FUNCTION_BLOCK FB_4PVICI_EPS EXTENDS FB_4PortViciValve
VAR_INPUT
END_VAR
VAR_OUTPUT
	bAllPortsLocked : BOOL;
	bExternalLock : BOOL;
END_VAR
VAR_IN_OUT
	aPortEPS : ARRAY [1 .. 4] OF DUT_VICI_PORT_EPS; // EPS for each port.
END_VAR
VAR
	{attribute 'pytmc' := '
	pv: PORT
	io: o
	'}
	iNewPortPos : INT;
	
	{attribute 'pytmc' := 'pv: OVRD_MODE'}
    bEPS_Override : BOOL := FALSE;
    {attribute 'pytmc' := 'pv: OVRD_COUNTDOWN'}
    tEPS_TimerCountDown : STRING := TIME_TO_STRING(T#0s);
    fbTimer : TON;
	tEPS_OVRD_RESET_TIME : TIME := T#1m;

	
END_VAR

iReqPos := LIMIT(1,iReqPos, 4); // KEEP EPS array index within bounds

M_RESET_OVERRIDE_TIMER();

iNewPortPos := M_EPS_LOGIC(aPortEPS := aPortEPS, 
							iReqPort := iReqPos,
							iPrevPort := iNewPortPos,
							bOverride := FALSE,
							bExternalLockSignal => bExternalLock,
							bAllPortsLocked => bAllPortsLocked);

fbNporValve(iAddress := iAdress, 
			iNumOfPorts := iNumPorts, 
			iReqPos := iNewPortPos);
			


(*
Qs
- Should there be a valve to stop the flow if none of the EPS conditions are met?
- Should the VICI valve always go to a EPS condition that is true?


PORT ENUM
- LOCKED 	(EPS not OK)
- UNLOCKED 	(EPS OK but not active)
- ACTIVE	(EPS OK and ACTIVE)
*)

METHOD M_EPS_LOGIC : INT
VAR_INPUT
	iReqPort : INT;
	iPrevPort : INT;
	bOverride : BOOL;
END_VAR
VAR_IN_OUT
	aPortEPS : ARRAY [1 .. 4] OF DUT_VICI_PORT_EPS;
END_VAR
VAR_OUTPUT
	bAllPortsLocked : BOOL;
	bExternalLockSignal : BOOL; // Signal to external device that port is locked.
END_VAR
VAR
	fbEPS : FB_EPS;
	iIndex : INT := 1;
	iEPS_NOT_OK_COUNT : INT;
	iNewPortPos : INT;
END_VAR
// Evaluate all EPS 
FOR iIndex := 1 TO iNumPorts BY 1 DO
	
	fbEPS(eps := aPortEPS[iIndex].stEPS);
	
	IF aPortEPS[iIndex].stEPS.bEPS_OK THEN
		aPortEPS[iIndex].ePortStatus := ENUM_PORT_STATUS.UNLOCKED;
	ELSE
		aPortEPS[iIndex].ePortStatus := ENUM_PORT_STATUS.LOCKED;
		iEPS_NOT_OK_COUNT := iEPS_NOT_OK_COUNT + 1;
	END_IF
	
END_FOR

iNewPortPos := iPrevPort;
IF aPortEPS[iReqPort].stEPS.bEPS_OK OR bOverride THEN
	aPortEPS[iReqPort].ePortStatus := ENUM_PORT_STATUS.ACTIVE;
	iNewPortPos := iReqPort;
END_IF

IF aPortEPS[iPrevPort].ePortStatus = ENUM_PORT_STATUS.LOCKED AND NOT bOverride THEN
	bExternalLockSignal := TRUE;
ELSIF aPortEPS[iPrevPort].ePortStatus <> ENUM_PORT_STATUS.LOCKED OR bOverride THEN
	bExternalLockSignal := FALSE;
END_IF

IF iEPS_NOT_OK_COUNT = iNumPorts AND NOT bOverride THEN
	bAllPortsLocked := TRUE;
ELSE
	bAllPortsLocked := FALSE;
END_IF

iEPS_NOT_OK_COUNT := 0;

M_EPS_LOGIC := iNewPortPos;
END_METHOD

METHOD M_RESET_OVERRIDE_TIMER
VAR_INPUT
END_VAR
fbTimer(IN := bEPS_Override, PT:= tEPS_OVRD_RESET_TIME);

IF bEPS_Override THEN
    tEPS_TimerCountDown := TIME_TO_STRING(tEPS_OVRD_RESET_TIME - fbTimer.ET);
END_IF

IF fbTimer.Q THEN
    bEPS_Override := FALSE;
    tEPS_TimerCountDown := TIME_TO_STRING(T#0s);
END_IF
END_METHOD

END_FUNCTION_BLOCK

(* stored: Version 1.1.0.1, ProductVersion 3.1.4024.12
   POU FB_4PVICI_EPS: Id {89dd5800-3edc-4db3-a7b8-40f2bc027efe}, SpecialFunc None
   Method M_EPS_LOGIC: Id {26579bdd-0757-429e-ab10-32602ebdd17d}
   Method M_RESET_OVERRIDE_TIMER: Id {ba020a30-4465-4930-9052-433997a4cf4f} *)
